(* Logix 5000 project; controller Modbus_TCP_Client_Example vendor 1 type 14 code 154 rev 32.15; software revision 32.05; part 2 of 10 *)

ADD_ON_INSTRUCTION AMP_Alarm_Reset_Servo   (* revision 1.0, vendor Applied Motion Products Inc. *)
// Applied Motion - Motor Alarm Reset - AOI
// Help:
// This AOI Reset Active Alarms(AX).
VAR_IN_OUT
   Input : DINT[20]; {required}   // Drive Input Assembly
   Output : DINT[11]; {required}   // Drive Output Assembly
        [10]   // Reserved
        [4]   // Target Velocity
        [0]   // Control Word
        [3]   // Target Pos
        [1]   // OpCode 1
        [2]   // OpCode 2
        [5]   // Porifle Acceleration
        [6]   // Profile Deceleration
        [7]   // Target Torque
        [8]   // OpCode 3
        [9]   // OpCode 4
END_VAR
VAR_INPUT
   Reset : BOOL; {required}   // Reset the Drive (on rising edge)
END_VAR
VAR_OUTPUT
   Sent : BOOL; {access Read Only, visible}   // Reset the Drive has been sent to drive
   In_Progress : BOOL; {access Read Only, visible}   // Reset in progress(not used)
   Done : BOOL; {access Read Only, visible}   // Reset completed without errors
   Error : BOOL; {access Read Only, visible}   // Reset failed
   State : DINT := 10; {access Read Only}   // Internal state of progress
END_VAR
VAR
   Loc_StatusCode : AMP_Status_Word_Servo; {access None}
   Loc_Reset_ONS : BOOL;
   Loc_Input_Assembly : AMP_Input_Assembly_Servo_v2; {access None}
   Loc_Command_Timeout : TIMER := (PRE := 2000); {access None}   // Timer to output fault if command is not Done
END_VAR

ROUTINE Logic   (* ladder *)
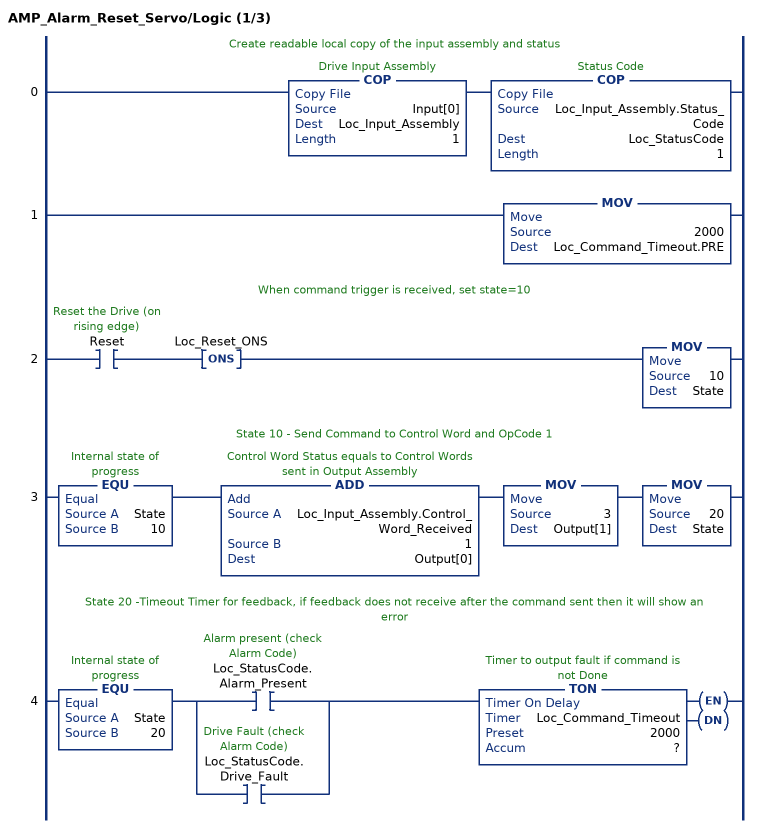
   // Create readable local copy of the input assembly and status
   0: COP(Input[0],Loc_Input_Assembly,1)COP(Loc_Input_Assembly.Status_Code,Loc_StatusCode,1);
   1: MOV(2000,Loc_Command_Timeout.PRE);
   // When command trigger is received, set state=10
   2: XIC(Reset)ONS(Loc_Reset_ONS)MOV(10,State);
   // State 10 - Send Command to Control Word and OpCode 1
   3: EQU(State,10)ADD(Loc_Input_Assembly.Control_Word_Received,1,Output[0])MOV(3,Output[1])MOV(20,State);
   // State 20 -Timeout Timer for feedback, if feedback does not receive after the command sent then it will show an error
   4: EQU(State,20)[XIC(Loc_StatusCode.Alarm_Present) ,XIC(Loc_StatusCode.Drive_Fault) ]TON(Loc_Command_Timeout,?,?);
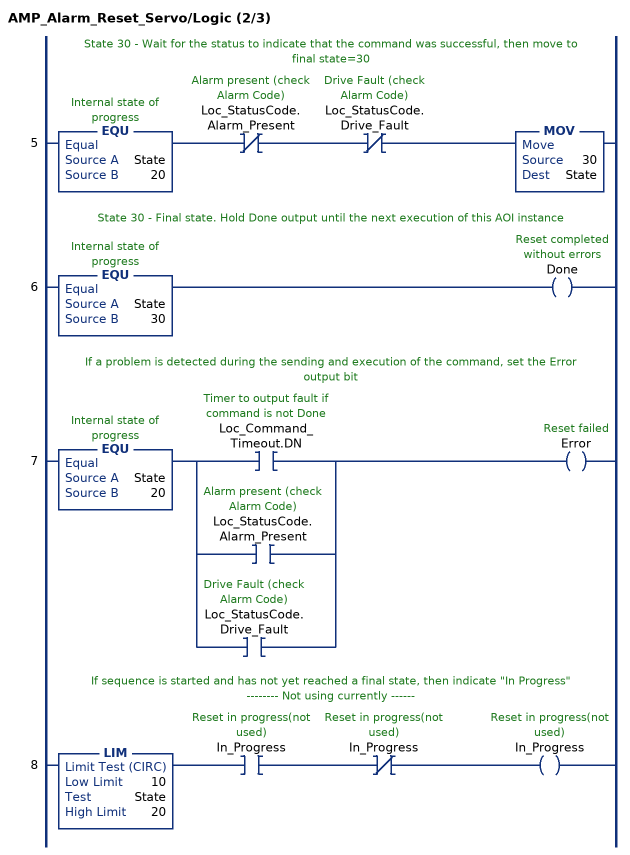
   // State 30 - Wait for the status to indicate that the command was successful, then move to final state=30
   5: EQU(State,20)XIO(Loc_StatusCode.Alarm_Present)XIO(Loc_StatusCode.Drive_Fault)MOV(30,State);
   // State 30 - Final state. Hold Done output until the next execution of this AOI instance
   6: EQU(State,30)OTE(Done);
   // If a problem is detected during the sending and execution of the command, set the Error output bit
   7: EQU(State,20)[XIC(Loc_Command_Timeout.DN) ,XIC(Loc_StatusCode.Alarm_Present) ,XIC(Loc_StatusCode.Drive_Fault) ]OTE(Error);
   // If sequence is started and has not yet reached a final state, then indicate "In Progress"
   // -------- Not using currently ------
   8: LIM(10,State,20)XIC(In_Progress)XIO(In_Progress)OTE(In_Progress);
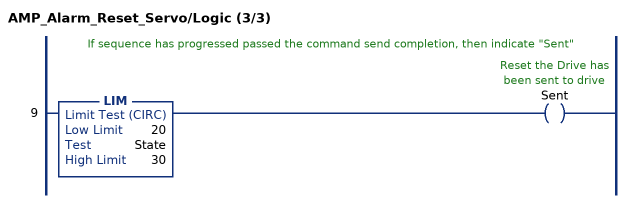
   // If sequence has progressed passed the command send completion, then indicate "Sent"
   9: LIM(20,State,30)OTE(Sent);
END_ROUTINE
END_ADD_ON_INSTRUCTION

ADD_ON_INSTRUCTION AMP_Crash_Stop_Servo   (* revision 1.0, vendor Applied Motion Products Inc. *)
// Applied Motion - Stop/Kill using Maximum Deceleration - AOI
// Help:
// This AOI immediately Stop the Motor Jogging/Moving(SK).
VAR_IN_OUT
   Input : DINT[20]; {required}   // Drive Input Assembly
        [4]   // Alarm_Code
        [16]   // Analog_Input1
        [0]   // Control_Word_Received
        [10]   // Position_Error
        [11]   // Actual_Velocity_RPS
        [12]   // Digital_Outputs
        [13]   // Digital_Inputs
        [14]   // Analog_Output1
        [15]   // Analog_Output2
        [17]   // Analog_Input2
        [18]   // Torque_Limit
        [19]   // Second_Encoder_Speed
        [1]   // OpCode1_Received
        [2]   // Control_Mode
        [3]   // Status_Code
        [5]   // Supply_Voltage
        [6]   // Applied_Torque
        [7]   // Drive_Temperature
        [8]   // Encoder_Position
        [9]   // Second_Encoder_Position
   Output : DINT[11]; {required}   // Drive Output Assembly
        [10]   // Reserved
        [4]   // Target Velocity
        [0]   // Control Word
        [3]   // Target Pos
        [1]   // OpCode 1
        [2]   // OpCode 2
        [5]   // Porifle Acceleration
        [6]   // Profile Deceleration
        [7]   // Target Torque
        [8]   // OpCode 3
        [9]   // OpCode 4
END_VAR
VAR_INPUT
   Stop : BOOL; {required}   // Crash Stop the drive axis (on rising edge)
END_VAR
VAR_OUTPUT
   Sent : BOOL; {access Read Only, visible}   // Stop has been sent to drive
   In_Progress : BOOL; {access Read Only, visible}   // Stop in progress
   Done : BOOL; {access Read Only, visible}   // Stop completed without errors - Servo is not moving
   Error : BOOL; {access Read Only, visible}   // Stop failed - drive not stopped or faulted
   State : DINT := 10; {access Read Only}   // Internal state of progress
END_VAR
VAR
   Loc_Stop_ONS : BOOL;
   Loc_StatusCode : AMP_Status_Word_Servo; {access None}
   Loc_Input_Assembly : AMP_Input_Assembly_Servo_v2; {access None}
END_VAR

ROUTINE Logic   (* ladder *)
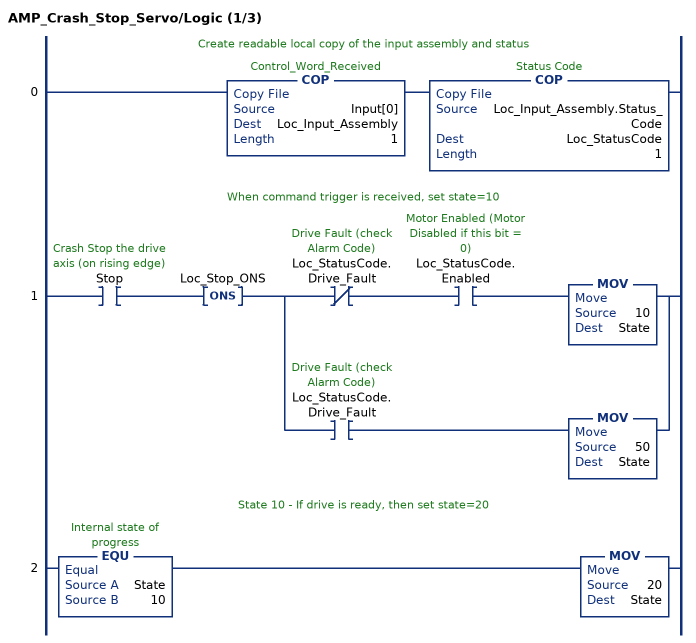
   // Create readable local copy of the input assembly and status
   0: COP(Input[0],Loc_Input_Assembly,1)COP(Loc_Input_Assembly.Status_Code,Loc_StatusCode,1);
   // When command trigger is received, set state=10
   1: XIC(Stop)ONS(Loc_Stop_ONS)[XIO(Loc_StatusCode.Drive_Fault) XIC(Loc_StatusCode.Enabled) MOV(10,State) ,XIC(Loc_StatusCode.Drive_Fault) MOV(50,State) ];
   // State 10 - If drive is ready, then set state=20
   2: EQU(State,10)MOV(20,State);
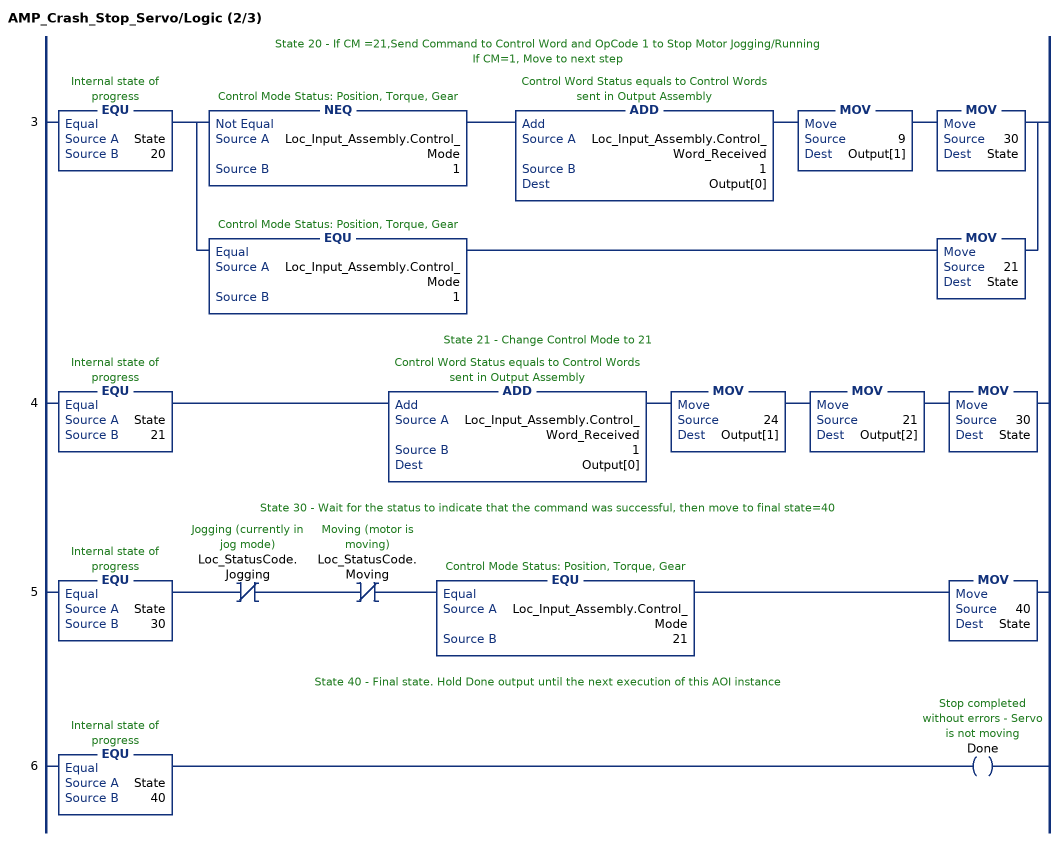
   // State 20 - If CM =21,Send Command to Control Word and OpCode 1 to Stop Motor Jogging/Running
   // If CM=1, Move to next step
   3: EQU(State,20)[NEQ(Loc_Input_Assembly.Control_Mode,1) ADD(Loc_Input_Assembly.Control_Word_Received,1,Output[0]) MOV(9,Output[1]) MOV(30,State) ,EQU(Loc_Input_Assembly.Control_Mode,1) MOV(21,State) ];
   // State 21 - Change Control Mode to 21
   4: EQU(State,21)ADD(Loc_Input_Assembly.Control_Word_Received,1,Output[0])MOV(24,Output[1])MOV(21,Output[2])MOV(30,State);
   // State 30 - Wait for the status to indicate that the command was successful, then move to final state=40
   5: EQU(State,30)XIO(Loc_StatusCode.Jogging)XIO(Loc_StatusCode.Moving)EQU(Loc_Input_Assembly.Control_Mode,21)MOV(40,State);
   // State 40 - Final state. Hold Done output until the next execution of this AOI instance
   6: EQU(State,40)OTE(Done);
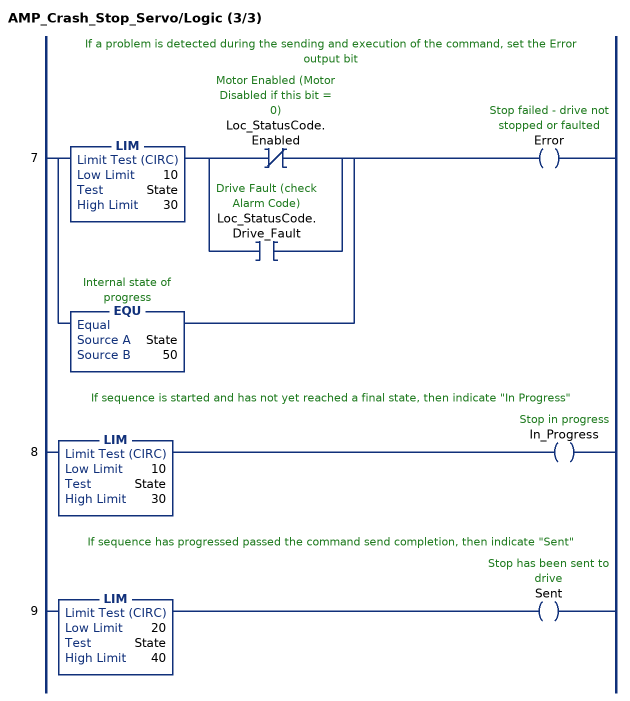
   // If a problem is detected during the sending and execution of the command, set the Error output bit
   7: [LIM(10,State,30) [XIO(Loc_StatusCode.Enabled) ,XIC(Loc_StatusCode.Drive_Fault) ] ,EQU(State,50) ]OTE(Error);
   // If sequence is started and has not yet reached a final state, then indicate "In Progress"
   8: LIM(10,State,30)OTE(In_Progress);
   // If sequence has progressed passed the command send completion, then indicate "Sent"
   9: LIM(20,State,40)OTE(Sent);
END_ROUTINE
END_ADD_ON_INSTRUCTION

ADD_ON_INSTRUCTION AMP_DI_Monitor_Servo   (* revision 1.0, vendor Applied Motion Products Inc. *)
// This AOI Monitor available Digital Input Status
// Help:
// Depending on which Drive/Motor Model you have, the number of IO Changes, Ignore extra IO monitoring
// 1 Represent Off/Open, 0 Represent On/Close
VAR_IN_OUT
   Input : DINT[20]; {required}   // Drive Input Assembly
END_VAR
VAR_OUTPUT
   DI_1 : BOOL; {visible}   // Digital Input 1, On = Input Opened, Off = Input Closed
   DI_2 : BOOL; {visible}   // Digital Input 2, On = Input Opened, Off = Input Closed
   DI_3 : BOOL; {visible}   // Digital Input 3, On = Input Opened, Off = Input Closed
   DI_4 : BOOL; {visible}   // Digital Input 4, On = Input Opened, Off = Input Closed
   DI_5 : BOOL; {visible}   // Digital Input 5, On = Input Opened, Off = Input Closed
   DI_6 : BOOL; {visible}   // Digital Input 6, On = Input Opened, Off = Input Closed
   DI_7 : BOOL; {visible}   // Digital Input 7, On = Input Opened, Off = Input Closed
   DI_8 : BOOL; {visible}   // Digital Input 8, On = Input Opened, Off = Input Closed
END_VAR
VAR
   Loc_StatusCode : AMP_Status_Word_Servo; {access None}
   Loc_Input_Assembly : AMP_Input_Assembly_Servo_v2; {access None}
   Inputs_DI : DINT; {access None}
END_VAR

ROUTINE Logic   (* ladder *)
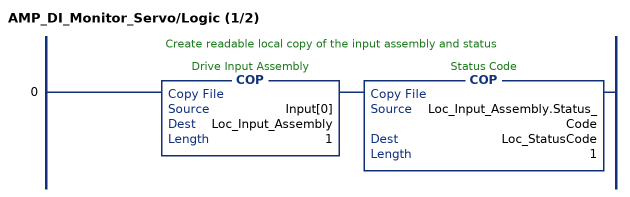
   // Create readable local copy of the input assembly and status
   0: COP(Input[0],Loc_Input_Assembly,1)COP(Loc_Input_Assembly.Status_Code,Loc_StatusCode,1);
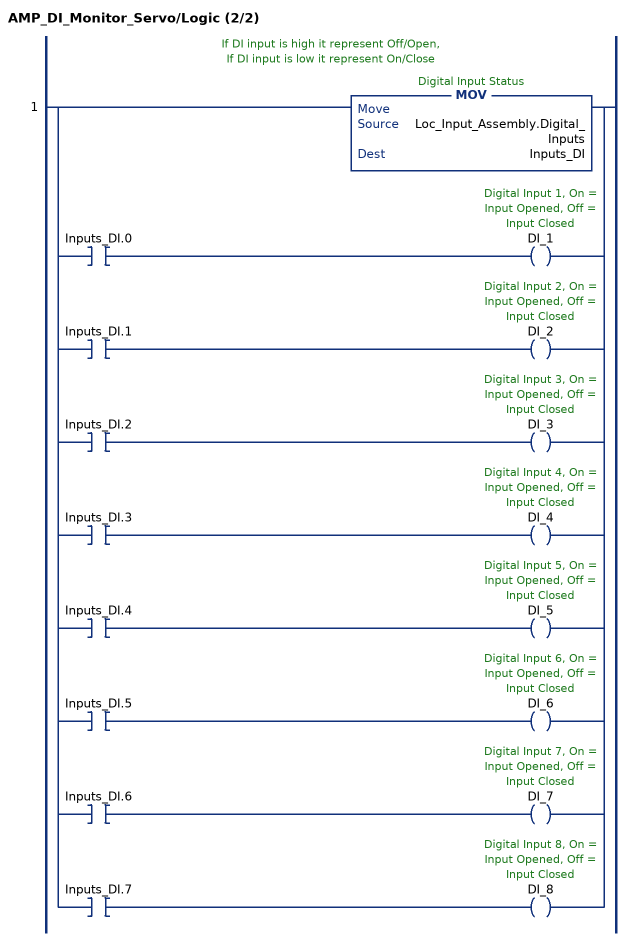
   // If DI input is high it represent Off/Open,
   // If DI input is low it represent On/Close
   1: [MOV(Loc_Input_Assembly.Digital_Inputs,Inputs_DI) ,XIC(Inputs_DI.0) OTE(DI_1) ,XIC(Inputs_DI.1) OTE(DI_2) ,XIC(Inputs_DI.2) OTE(DI_3) ,XIC(Inputs_DI.3) OTE(DI_4) ,XIC(Inputs_DI.4) OTE(DI_5) ,XIC(Inputs_DI.5) OTE(DI_6) ,XIC(Inputs_DI.6) OTE(DI_7) ,XIC(Inputs_DI.7) OTE(DI_8) ];
END_ROUTINE
END_ADD_ON_INSTRUCTION

ADD_ON_INSTRUCTION AMP_DO_Control_Servo   (* revision 1.0, vendor Applied Motion Products Inc. *)
// Applied Motion - General Purpose Digital Output Control - AOI
// Help:
// This AOI only Controls Output that are defined as General Purpose Output.
// Depending on which Drive/Motor Model you have, the number of Output Changes, Ignore extra Output.
// Define output number 1-6 and Condition L to Close the output, H to Open the Output.
// As an example, 2L will set output number 2 Close.
// This AOI can be used when Motor is Enable or Disable.
VAR_IN_OUT
   Input : DINT[20]; {required}   // Drive Input Assembly
        [16]   // Analog_Input1
        [4]   // Alarm_Code
        [0]   // Control_Word_Received
        [10]   // Position_Error
        [11]   // Actual_Velocity_RPS
        [12]   // Digital_Outputs
        [13]   // Digital_Inputs
        [14]   // Analog_Output1
        [15]   // Analog_Output2
        [17]   // Analog_Input2
        [18]   // Torque_Limit
        [19]   // Second_Encoder_Speed
        [1]   // OpCode1_Received
        [2]   // Control_Mode
        [3]   // Status_Code
        [5]   // Supply_Voltage
        [6]   // Applied_Torque
        [7]   // Drive_Temperature
        [8]   // Encoder_Position
        [9]   // Second_Encoder_Position
   Output : DINT[11]; {required}   // Drive Output Assembly
        [10]   // Reserved
        [4]   // Target Velocity
        [0]   // Control Word
        [3]   // Target Pos
        [1]   // OpCode 1
        [2]   // OpCode 2
        [5]   // Porifle Acceleration
        [6]   // Profile Deceleration
        [7]   // Target Torque
        [8]   // OpCode 3
        [9]   // OpCode 4
END_VAR
VAR_INPUT
   Execute : BOOL; {required}   // Execute the SCL command 'SO'
   Output_Number : INT; {required}   // Output Number, 1-6
   Condition : SINT; {required}   // Output Condition: H for Open and L for Close Output
END_VAR
VAR_OUTPUT
   DO_1 : BOOL; {visible}   // Digital Output 1, On = Output Closed, Off = Output Opened
   DO_2 : BOOL; {visible}   // Digital Output 2, On = Output Closed, Off = Output Opened
   DO_3 : BOOL; {visible}   // Digital Output 3, On = Output Closed, Off = Output Opened
   DO_4 : BOOL; {visible}   // Digital Output 4, On = Output Closed, Off = Output Opened
   DO_5 : BOOL; {visible}   // Digital Output 5, On = Output Closed, Off = Output Opened
   DO_6 : BOOL; {visible}   // Digital Output 6, On = Output Closed, Off = Output Opened
END_VAR
VAR
   Loc_StatusCode : AMP_Status_Word_Servo;
   Loc_Input_Assembly : AMP_Input_Assembly_Servo_v2;
   Loc_SCL_ONS : BOOL;
   Loc_Outputs_DO : INT; {access None}
   Loc_IO_Condition_Encoded : DINT; {access None}
   Loc_IO1_Number_Encoded : DINT; {access None}
   Loc_State : DINT := 10; {access Read Only}   // Internal state of progress
   Loc_Error : BOOL; {access Read Only}   // Command failed
   Loc_Done : BOOL; {access Read Only}   // Command completed without errors - Drive is Homed
   Loc_In_Progress : BOOL; {access Read Only}   // Command in progress
   Loc_Sent : BOOL; {access Read Only}   // Command has sent
END_VAR

ROUTINE Logic   (* ladder *)
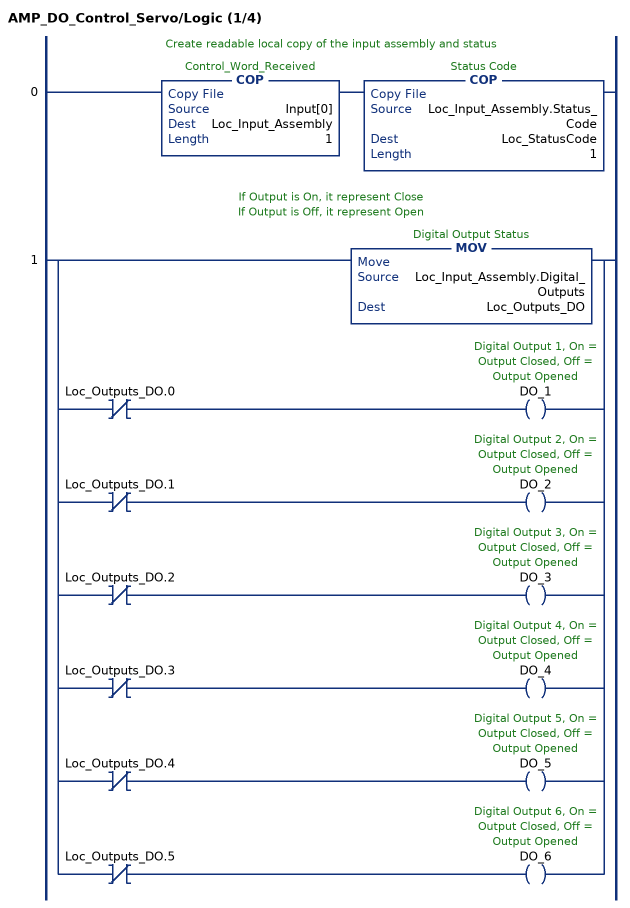
   // Create readable local copy of the input assembly and status
   0: COP(Input[0],Loc_Input_Assembly,1)COP(Loc_Input_Assembly.Status_Code,Loc_StatusCode,1);
   // If Output is On, it represent Close
   // If Output is Off, it represent Open
   1: [MOV(Loc_Input_Assembly.Digital_Outputs,Loc_Outputs_DO) ,XIO(Loc_Outputs_DO.0) OTE(DO_1) ,XIO(Loc_Outputs_DO.1) OTE(DO_2) ,XIO(Loc_Outputs_DO.2) OTE(DO_3) ,XIO(Loc_Outputs_DO.3) OTE(DO_4) ,XIO(Loc_Outputs_DO.4) OTE(DO_5) ,XIO(Loc_Outputs_DO.5) OTE(DO_6) ];
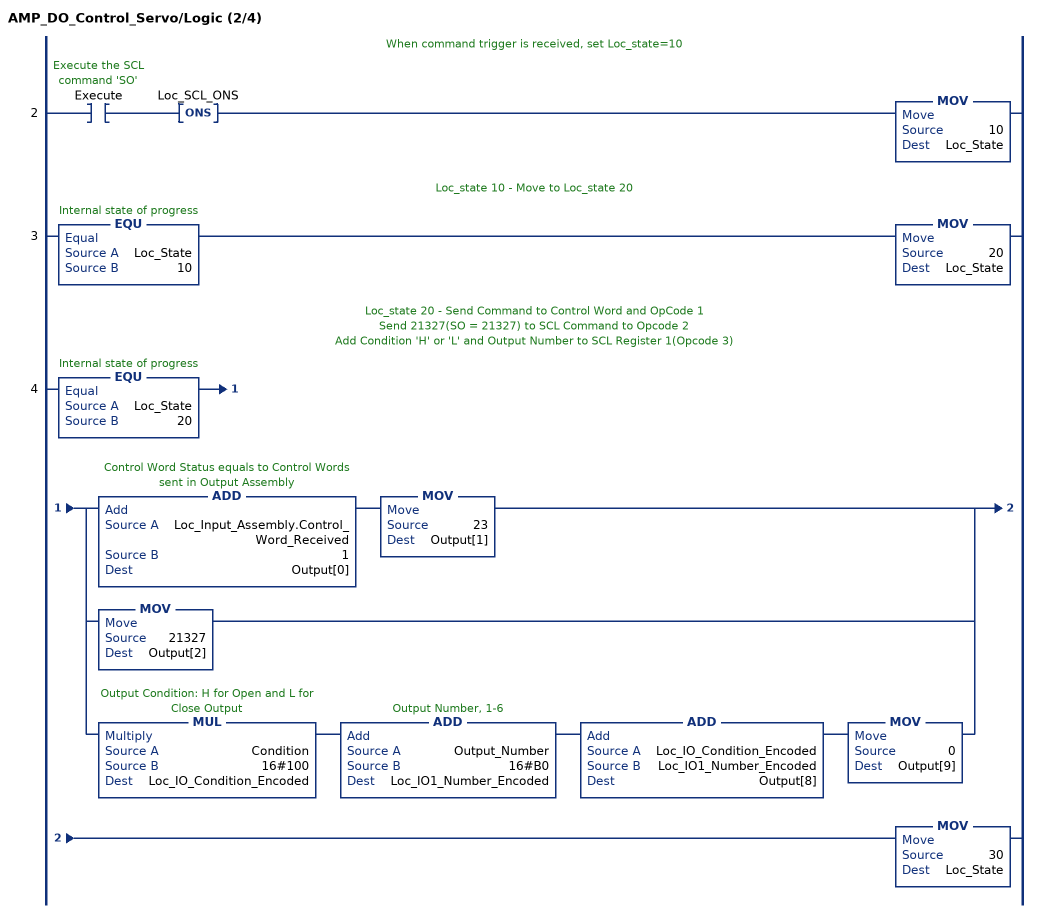
   // When command trigger is received, set Loc_state=10
   2: XIC(Execute)ONS(Loc_SCL_ONS)MOV(10,Loc_State);
   // Loc_state 10 - Move to Loc_state 20
   3: EQU(Loc_State,10)MOV(20,Loc_State);
   // Loc_state 20 - Send Command to Control Word and OpCode 1
   // Send 21327(SO = 21327) to SCL Command to Opcode 2
   // Add Condition 'H' or 'L' and Output Number to SCL Register 1(Opcode 3)
   4: EQU(Loc_State,20)[ADD(Loc_Input_Assembly.Control_Word_Received,1,Output[0]) MOV(23,Output[1]) ,MOV(21327,Output[2]) ,MUL(Condition,16#100,Loc_IO_Condition_Encoded) ADD(Output_Number,16#B0,Loc_IO1_Number_Encoded) ADD(Loc_IO_Condition_Encoded,Loc_IO1_Number_Encoded,Output[8]) MOV(0,Output[9]) ]MOV(30,Loc_State);
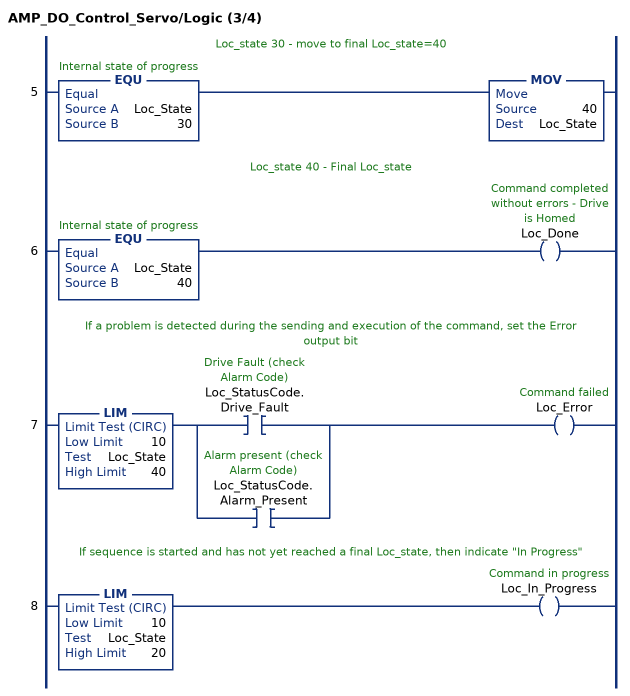
   // Loc_state 30 - move to final Loc_state=40
   5: EQU(Loc_State,30)MOV(40,Loc_State);
   // Loc_state 40 - Final Loc_state
   6: EQU(Loc_State,40)OTE(Loc_Done);
   // If a problem is detected during the sending and execution of the command, set the Error output bit
   7: LIM(10,Loc_State,40)[XIC(Loc_StatusCode.Drive_Fault) ,XIC(Loc_StatusCode.Alarm_Present) ]OTE(Loc_Error);
   // If sequence is started and has not yet reached a final Loc_state, then indicate "In Progress"
   8: LIM(10,Loc_State,20)OTE(Loc_In_Progress);
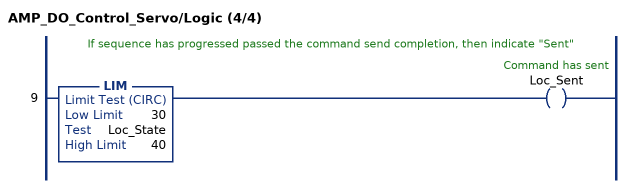
   // If sequence has progressed passed the command send completion, then indicate "Sent"
   9: LIM(30,Loc_State,40)OTE(Loc_Sent);
END_ROUTINE
END_ADD_ON_INSTRUCTION

ADD_ON_INSTRUCTION AMP_Hard_Stop_Homing   (* revision 1.0 *)
// Applied Motion - Hard Stop Homing AOI
// Help:
// The Hard Stop Homing AOI accepts all the required parameters for SCL commands HV1, HV2, HV3, HA1, HA2, HA3, HL1, HL2, HL3, HC, HD, HO and then sends the HS command to initiate the Hard Stop Homing move.
VAR_IN_OUT
   Input : DINT[14]; {required}   // Drive Input Assembly
   Output : DINT[16]; {required}   // Drive Output Assembly
        [0]   // Command Word
        [10]   // Data/Register 1
        [11]   // Data/Register 2
        [1]   // Jog Speed (0.25 rev/min)
        [2]   // Jog Acceleration (10 rev/s/s)
        [3]   // Jog Deceleration (10 rev/s/s)
        [4]   // Point-to-Point Velocity (0.25 rev/min)
        [5]   // Point-to-Point Acceleration (10 rev/s/s)
        [6]   // Point-to-Point Deceleration (10 rev/s/s)
        [7]   // Point-to-Point Distance (Motor steps)
        [9]   // (2x ASCII Letters in 16 lower word)
END_VAR
VAR_INPUT
   RPI : DINT := 100; {visible}   // Drive Connection Request Packet Interval (milliseconds)
   Start : BOOL; {required}   // Start the Homing
   HV1 : REAL; {required}   // Velocity used while seeking the hard stop (rev/s)
   HV2 : REAL; {required}   // Velocity when moving offset distance set by HO (rev/s)
   HV3 : REAL; {required}   // Velocity when searching for encoder index if desired (rev/s)
   HA1 : REAL; {required}   // Accel used while seeking the hard stop (rev/s/s)
   HA2 : REAL; {required}   // Accel when moving offset distance set by HO (rev/s/s)
   HA3 : REAL; {required}   // Accel when searching for encoder index if desired (rev/s/s)
   HL1 : REAL; {required}   // Decel used while seeking the hard stop (rev/s/s)
   HL2 : REAL; {required}   // Decel when moving offset distance set by HO (rev/s/s)
   HL3 : REAL; {required}   // Decel when searching for encoder index if desired (rev/s/s)
   HC : REAL; {required}   // Hard Stop Current (Amps)
   HD : DINT; {required}   // Hard Stop Fault Delay (ms)
   HO : DINT; {required}   // Home Offset (steps, negative = CCW, positive = CW)
   HS : DINT; {required}   // Hard Stop method (0 = without index, 1 = with index)
END_VAR
VAR_OUTPUT
   Sent : BOOL; {access Read Only, visible}   // All parameter setting and homing commands have been sent to drive
   In_Progress : BOOL; {access Read Only, visible}   // The setting of parameters and/or homing are in progress
   Done : BOOL; {access Read Only, visible}   // Homing Move completed without errors - desired position reached
   Error : BOOL; {access Read Only, visible}   // Homing failed to complete - drive not ready or faulted
   State : DINT := 34; {access Read Only}   // Internal state of progress
END_VAR
VAR
   Loc_StatusCode : AMP_Status_Word;
   Loc_CommandOff_Timer : TIMER;   // Timer to make sure command value was 0 before sending a new command
   Loc_CommandOn_Timer : TIMER;   // Timer to make sure command value is set long enough to be sent to drive
   Loc_Input_Assembly : AMP_Input_Assembly_v2; {access None}
   Loc_Start_ONS : BOOL; {access None}
END_VAR

ROUTINE Logic   (* ladder *)
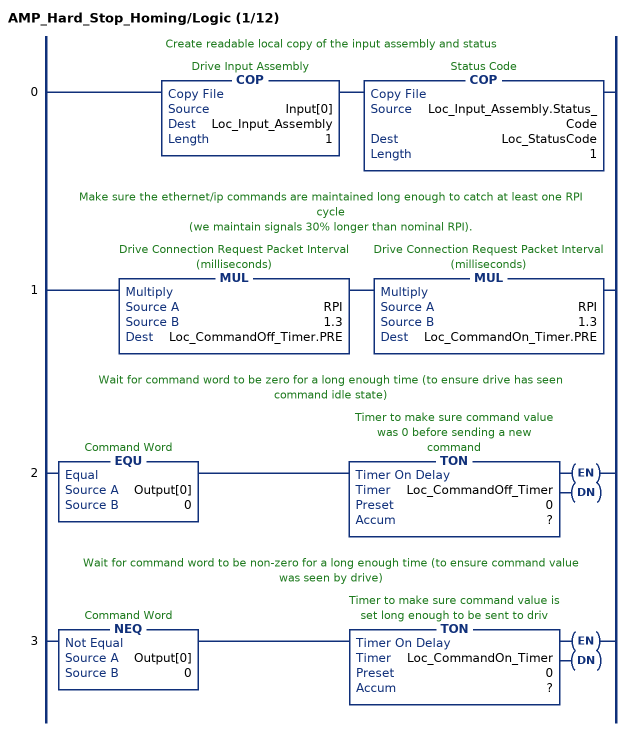
   // Create readable local copy of the input assembly and status
   0: COP(Input[0],Loc_Input_Assembly,1)COP(Loc_Input_Assembly.Status_Code,Loc_StatusCode,1);
   // Make sure the ethernet/ip commands are maintained long enough to catch at least one RPI cycle
   // (we maintain signals 30% longer than nominal RPI).
   1: MUL(RPI,1.3,Loc_CommandOff_Timer.PRE)MUL(RPI,1.3,Loc_CommandOn_Timer.PRE);
   // Wait for command word to be zero for a long enough time (to ensure drive has seen command idle state)
   2: EQU(Output[0],0)TON(Loc_CommandOff_Timer,?,?);
   // Wait for command word to be non-zero for a long enough time (to ensure command value was seen by drive)
   3: NEQ(Output[0],0)TON(Loc_CommandOn_Timer,?,?);
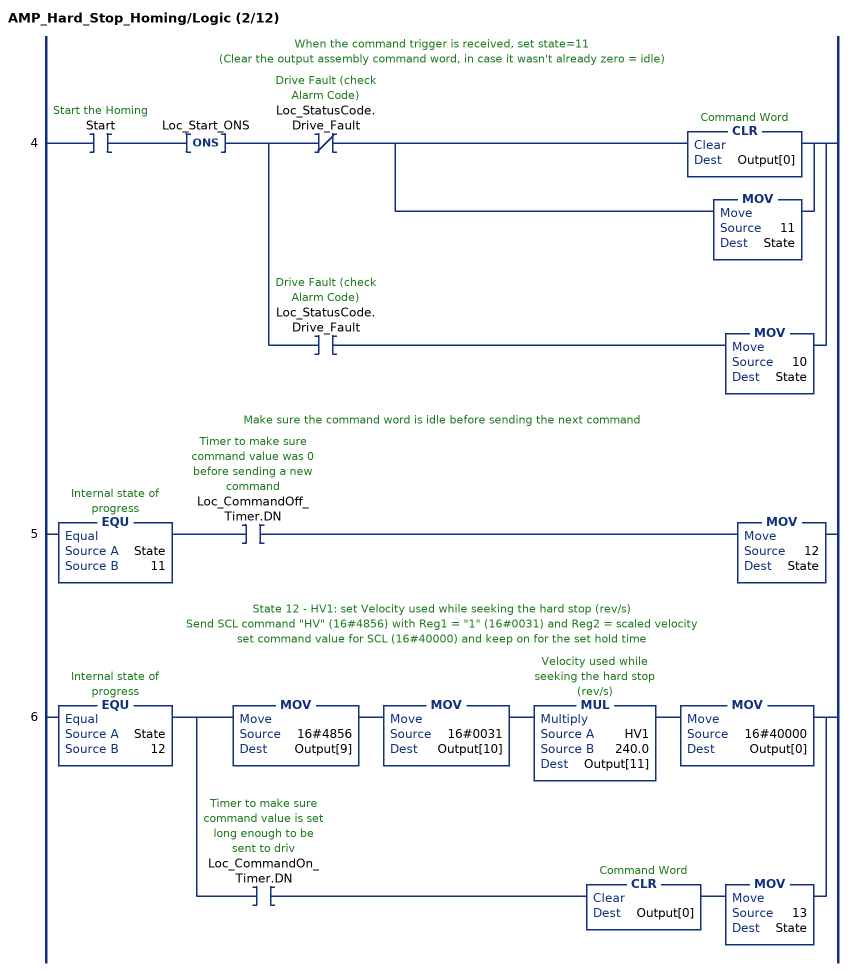
   // When the command trigger is received, set state=11
   // (Clear the output assembly command word, in case it wasn't already zero = idle)
   4: XIC(Start)ONS(Loc_Start_ONS)[XIO(Loc_StatusCode.Drive_Fault) [CLR(Output[0]) ,MOV(11,State) ] ,XIC(Loc_StatusCode.Drive_Fault) MOV(10,State) ];
   // Make sure the command word is idle before sending the next command
   5: EQU(State,11)XIC(Loc_CommandOff_Timer.DN)MOV(12,State);
   // State 12 - HV1: set Velocity used while seeking the hard stop (rev/s)
   // Send SCL command "HV" (16#4856) with Reg1 = "1" (16#0031) and Reg2 = scaled velocity
   // set command value for SCL (16#40000) and keep on for the set hold time
   6: EQU(State,12)[MOV(16#4856,Output[9]) MOV(16#0031,Output[10]) MUL(HV1,240.0,Output[11]) MOV(16#40000,Output[0]) ,XIC(Loc_CommandOn_Timer.DN) CLR(Output[0]) MOV(13,State) ];
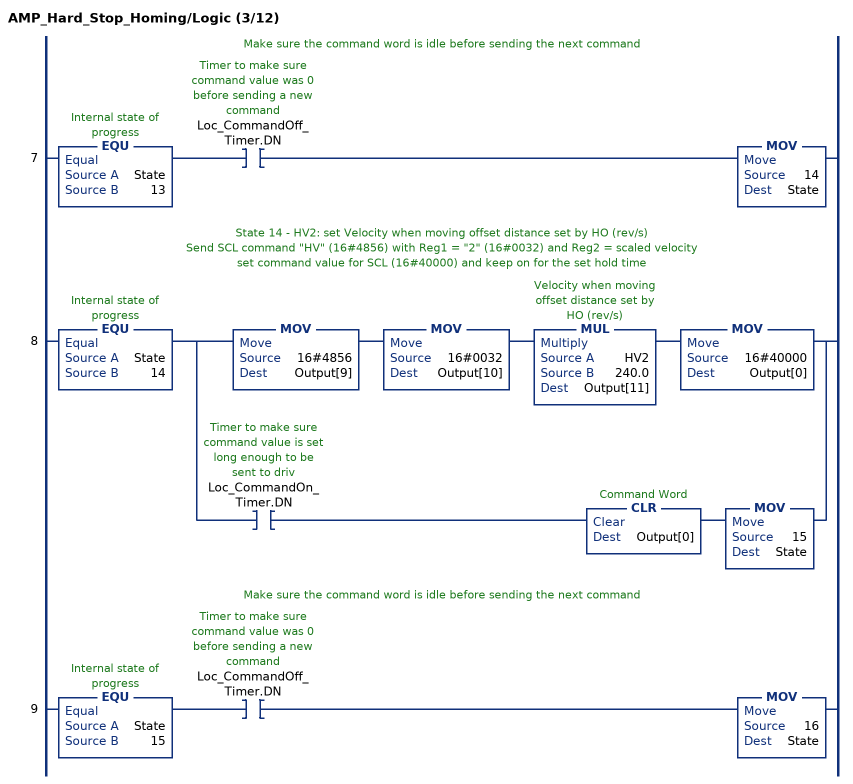
   // Make sure the command word is idle before sending the next command
   7: EQU(State,13)XIC(Loc_CommandOff_Timer.DN)MOV(14,State);
   // State 14 - HV2: set Velocity when moving offset distance set by HO (rev/s)
   // Send SCL command "HV" (16#4856) with Reg1 = "2" (16#0032) and Reg2 = scaled velocity
   // set command value for SCL (16#40000) and keep on for the set hold time
   8: EQU(State,14)[MOV(16#4856,Output[9]) MOV(16#0032,Output[10]) MUL(HV2,240.0,Output[11]) MOV(16#40000,Output[0]) ,XIC(Loc_CommandOn_Timer.DN) CLR(Output[0]) MOV(15,State) ];
   // Make sure the command word is idle before sending the next command
   9: EQU(State,15)XIC(Loc_CommandOff_Timer.DN)MOV(16,State);
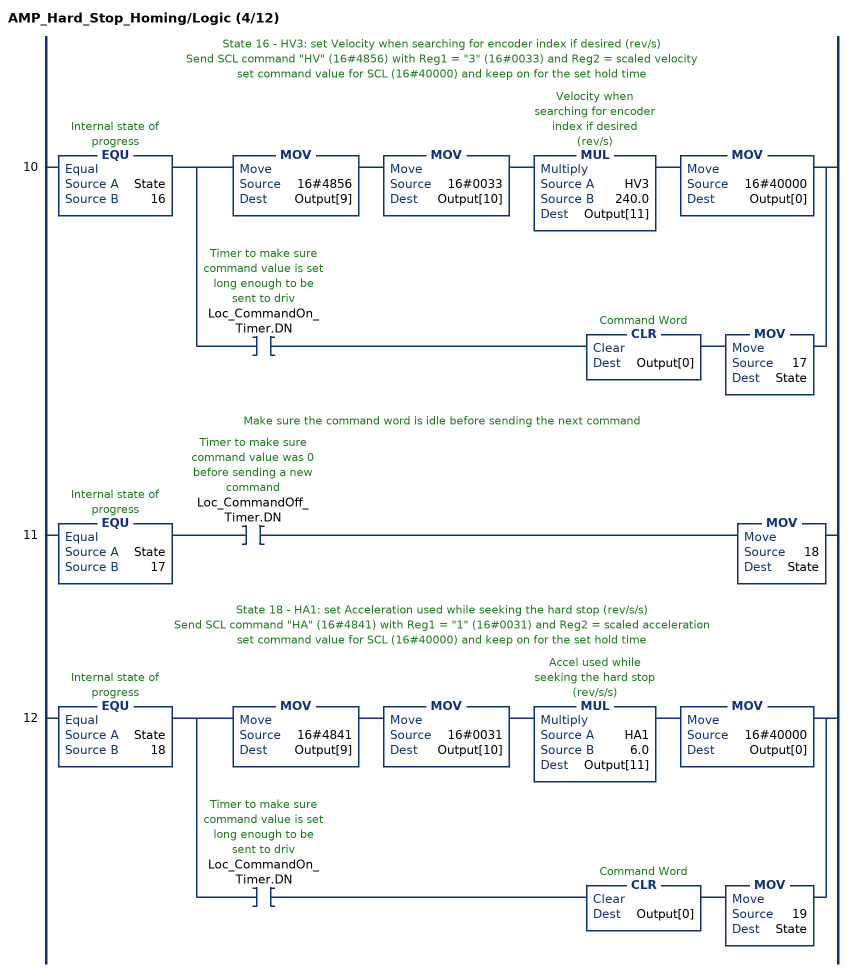
   // State 16 - HV3: set Velocity when searching for encoder index if desired (rev/s)
   // Send SCL command "HV" (16#4856) with Reg1 = "3" (16#0033) and Reg2 = scaled velocity
   // set command value for SCL (16#40000) and keep on for the set hold time
   10: EQU(State,16)[MOV(16#4856,Output[9]) MOV(16#0033,Output[10]) MUL(HV3,240.0,Output[11]) MOV(16#40000,Output[0]) ,XIC(Loc_CommandOn_Timer.DN) CLR(Output[0]) MOV(17,State) ];
   // Make sure the command word is idle before sending the next command
   11: EQU(State,17)XIC(Loc_CommandOff_Timer.DN)MOV(18,State);
   // State 18 - HA1: set Acceleration used while seeking the hard stop (rev/s/s)
   // Send SCL command "HA" (16#4841) with Reg1 = "1" (16#0031) and Reg2 = scaled acceleration
   // set command value for SCL (16#40000) and keep on for the set hold time
   12: EQU(State,18)[MOV(16#4841,Output[9]) MOV(16#0031,Output[10]) MUL(HA1,6.0,Output[11]) MOV(16#40000,Output[0]) ,XIC(Loc_CommandOn_Timer.DN) CLR(Output[0]) MOV(19,State) ];
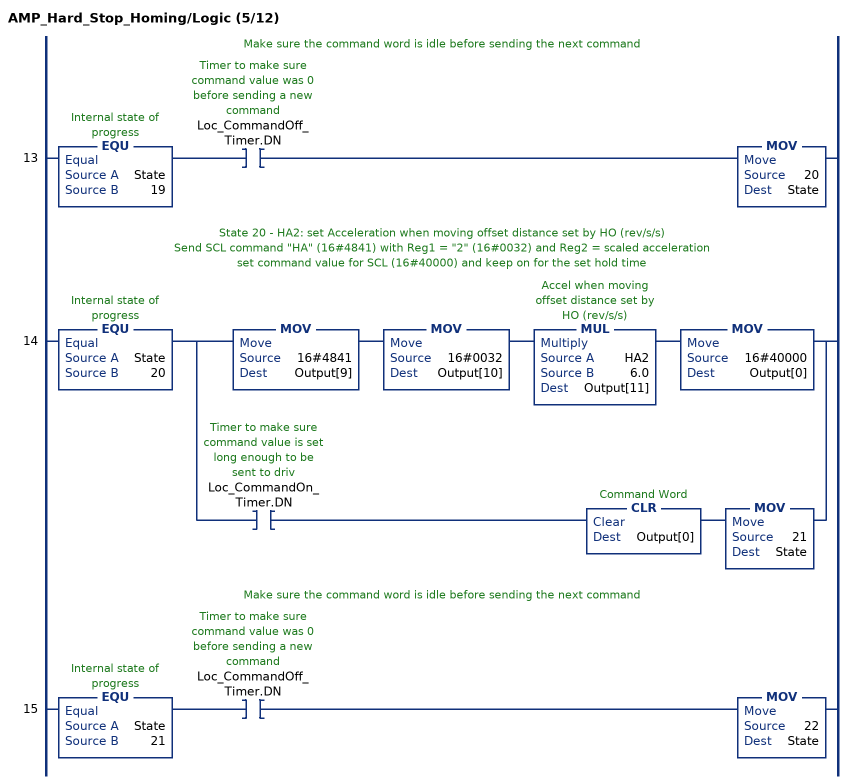
   // Make sure the command word is idle before sending the next command
   13: EQU(State,19)XIC(Loc_CommandOff_Timer.DN)MOV(20,State);
   // State 20 - HA2: set Acceleration when moving offset distance set by HO (rev/s/s)
   // Send SCL command "HA" (16#4841) with Reg1 = "2" (16#0032) and Reg2 = scaled acceleration
   // set command value for SCL (16#40000) and keep on for the set hold time
   14: EQU(State,20)[MOV(16#4841,Output[9]) MOV(16#0032,Output[10]) MUL(HA2,6.0,Output[11]) MOV(16#40000,Output[0]) ,XIC(Loc_CommandOn_Timer.DN) CLR(Output[0]) MOV(21,State) ];
   // Make sure the command word is idle before sending the next command
   15: EQU(State,21)XIC(Loc_CommandOff_Timer.DN)MOV(22,State);
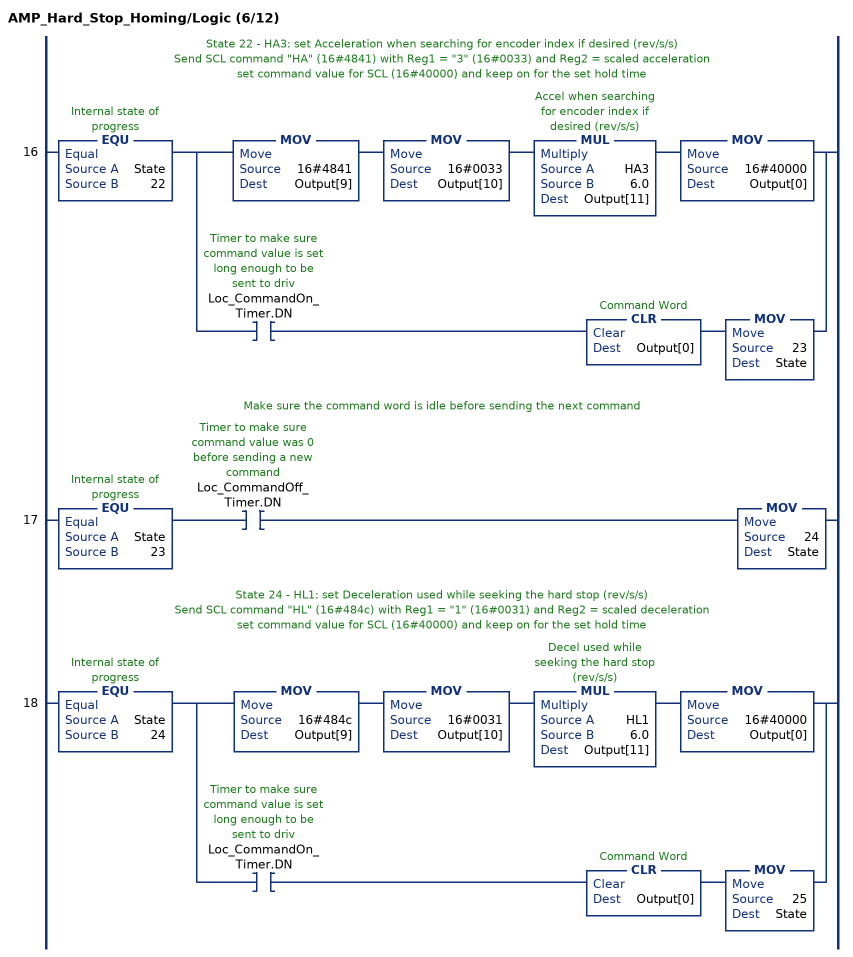
   // State 22 - HA3: set Acceleration when searching for encoder index if desired (rev/s/s)
   // Send SCL command "HA" (16#4841) with Reg1 = "3" (16#0033) and Reg2 = scaled acceleration
   // set command value for SCL (16#40000) and keep on for the set hold time
   16: EQU(State,22)[MOV(16#4841,Output[9]) MOV(16#0033,Output[10]) MUL(HA3,6.0,Output[11]) MOV(16#40000,Output[0]) ,XIC(Loc_CommandOn_Timer.DN) CLR(Output[0]) MOV(23,State) ];
   // Make sure the command word is idle before sending the next command
   17: EQU(State,23)XIC(Loc_CommandOff_Timer.DN)MOV(24,State);
   // State 24 - HL1: set Deceleration used while seeking the hard stop (rev/s/s)
   // Send SCL command "HL" (16#484c) with Reg1 = "1" (16#0031) and Reg2 = scaled deceleration
   // set command value for SCL (16#40000) and keep on for the set hold time
   18: EQU(State,24)[MOV(16#484c,Output[9]) MOV(16#0031,Output[10]) MUL(HL1,6.0,Output[11]) MOV(16#40000,Output[0]) ,XIC(Loc_CommandOn_Timer.DN) CLR(Output[0]) MOV(25,State) ];
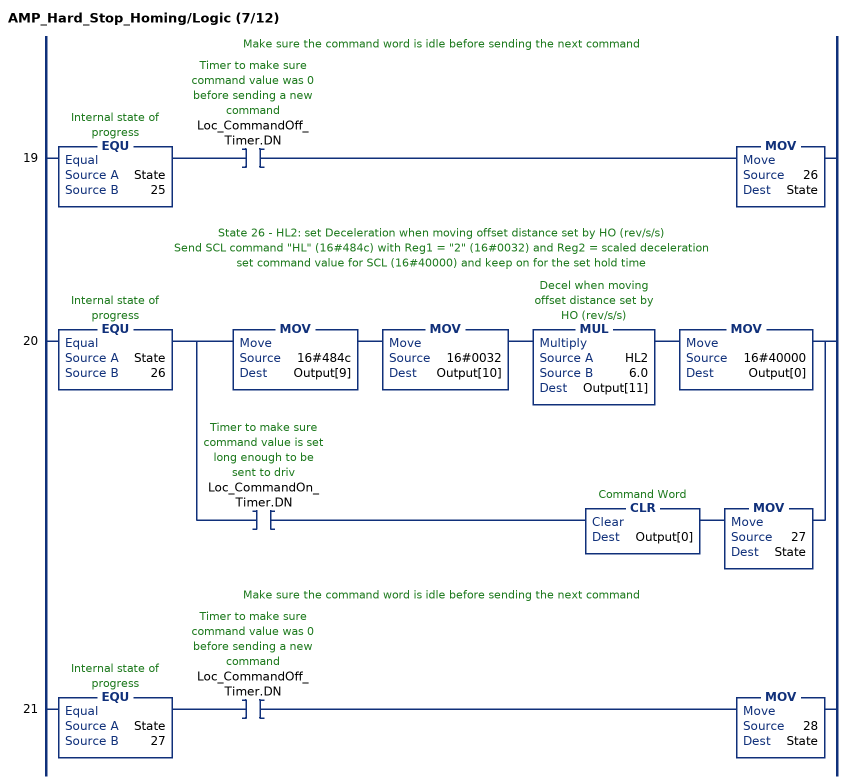
   // Make sure the command word is idle before sending the next command
   19: EQU(State,25)XIC(Loc_CommandOff_Timer.DN)MOV(26,State);
   // State 26 - HL2: set Deceleration when moving offset distance set by HO (rev/s/s)
   // Send SCL command "HL" (16#484c) with Reg1 = "2" (16#0032) and Reg2 = scaled deceleration
   // set command value for SCL (16#40000) and keep on for the set hold time
   20: EQU(State,26)[MOV(16#484c,Output[9]) MOV(16#0032,Output[10]) MUL(HL2,6.0,Output[11]) MOV(16#40000,Output[0]) ,XIC(Loc_CommandOn_Timer.DN) CLR(Output[0]) MOV(27,State) ];
   // Make sure the command word is idle before sending the next command
   21: EQU(State,27)XIC(Loc_CommandOff_Timer.DN)MOV(28,State);
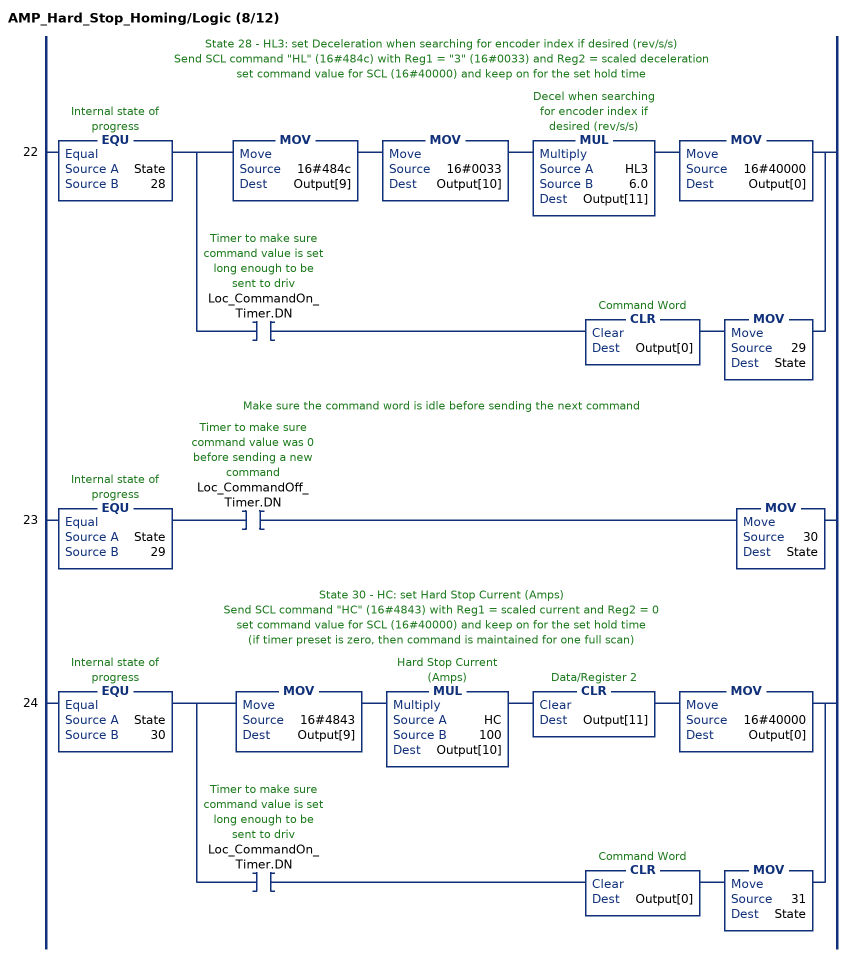
   // State 28 - HL3: set Deceleration when searching for encoder index if desired (rev/s/s)
   // Send SCL command "HL" (16#484c) with Reg1 = "3" (16#0033) and Reg2 = scaled deceleration
   // set command value for SCL (16#40000) and keep on for the set hold time
   22: EQU(State,28)[MOV(16#484c,Output[9]) MOV(16#0033,Output[10]) MUL(HL3,6.0,Output[11]) MOV(16#40000,Output[0]) ,XIC(Loc_CommandOn_Timer.DN) CLR(Output[0]) MOV(29,State) ];
   // Make sure the command word is idle before sending the next command
   23: EQU(State,29)XIC(Loc_CommandOff_Timer.DN)MOV(30,State);
   // State 30 - HC: set Hard Stop Current (Amps)
   // Send SCL command "HC" (16#4843) with Reg1 = scaled current and Reg2 = 0
   // set command value for SCL (16#40000) and keep on for the set hold time
   // (if timer preset is zero, then command is maintained for one full scan)
   24: EQU(State,30)[MOV(16#4843,Output[9]) MUL(HC,100,Output[10]) CLR(Output[11]) MOV(16#40000,Output[0]) ,XIC(Loc_CommandOn_Timer.DN) CLR(Output[0]) MOV(31,State) ];
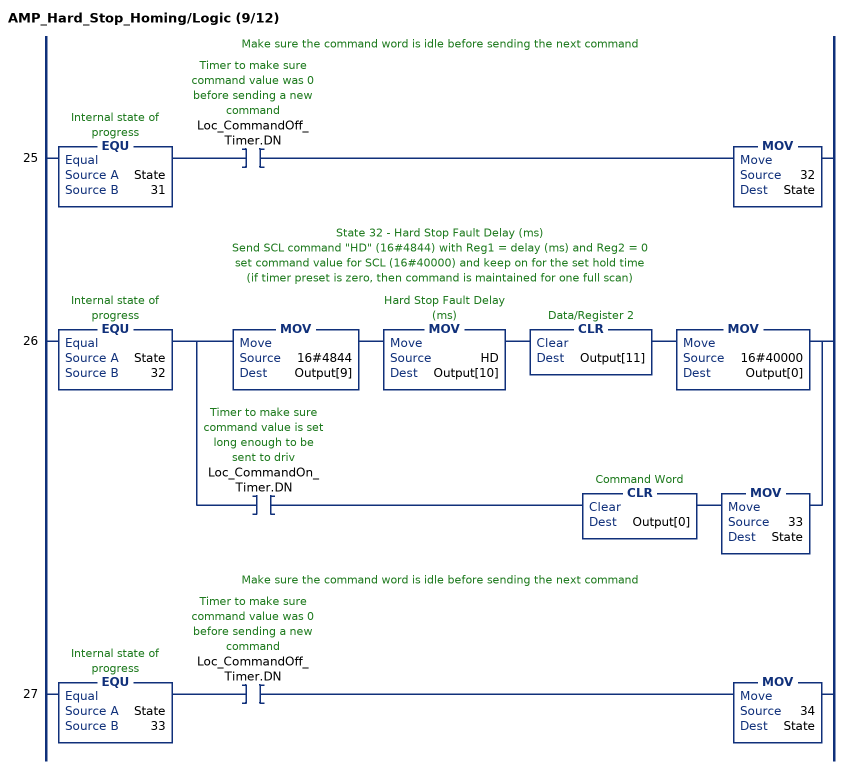
   // Make sure the command word is idle before sending the next command
   25: EQU(State,31)XIC(Loc_CommandOff_Timer.DN)MOV(32,State);
   // State 32 - Hard Stop Fault Delay (ms)
   // Send SCL command "HD" (16#4844) with Reg1 = delay (ms) and Reg2 = 0
   // set command value for SCL (16#40000) and keep on for the set hold time
   // (if timer preset is zero, then command is maintained for one full scan)
   26: EQU(State,32)[MOV(16#4844,Output[9]) MOV(HD,Output[10]) CLR(Output[11]) MOV(16#40000,Output[0]) ,XIC(Loc_CommandOn_Timer.DN) CLR(Output[0]) MOV(33,State) ];
   // Make sure the command word is idle before sending the next command
   27: EQU(State,33)XIC(Loc_CommandOff_Timer.DN)MOV(34,State);
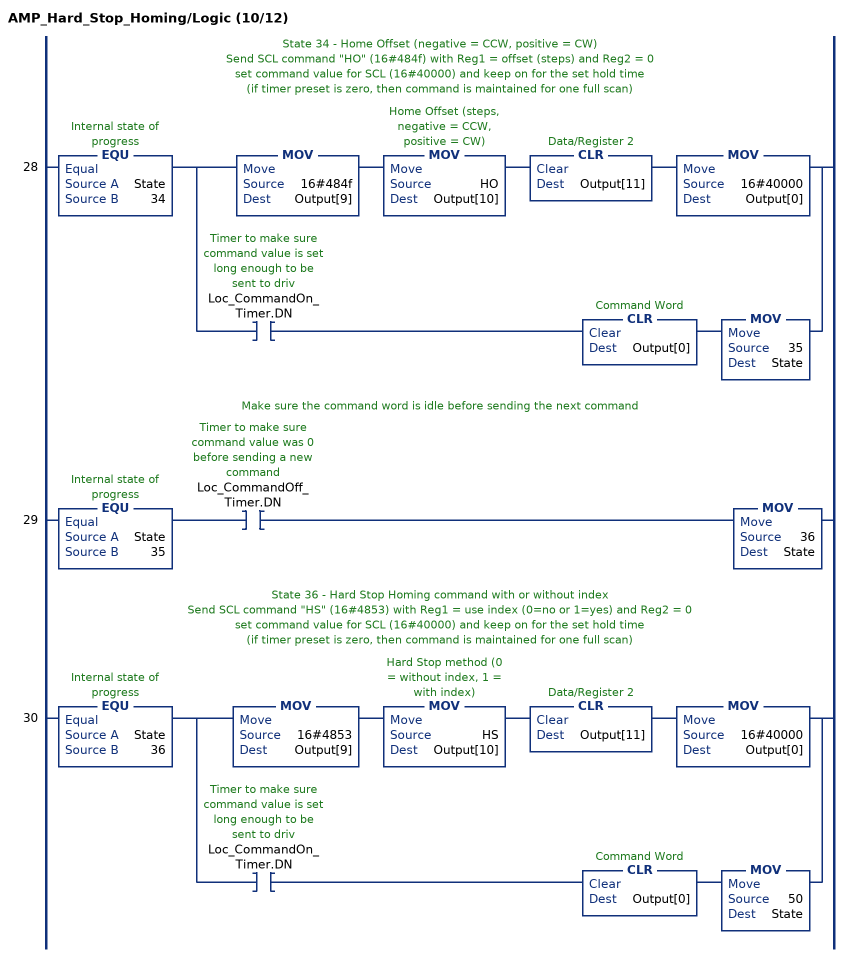
   // State 34 - Home Offset (negative = CCW, positive = CW)
   // Send SCL command "HO" (16#484f) with Reg1 = offset (steps) and Reg2 = 0
   // set command value for SCL (16#40000) and keep on for the set hold time
   // (if timer preset is zero, then command is maintained for one full scan)
   28: EQU(State,34)[MOV(16#484f,Output[9]) MOV(HO,Output[10]) CLR(Output[11]) MOV(16#40000,Output[0]) ,XIC(Loc_CommandOn_Timer.DN) CLR(Output[0]) MOV(35,State) ];
   // Make sure the command word is idle before sending the next command
   29: EQU(State,35)XIC(Loc_CommandOff_Timer.DN)MOV(36,State);
   // State 36 - Hard Stop Homing command with or without index
   // Send SCL command "HS" (16#4853) with Reg1 = use index (0=no or 1=yes) and Reg2 = 0
   // set command value for SCL (16#40000) and keep on for the set hold time
   // (if timer preset is zero, then command is maintained for one full scan)
   30: EQU(State,36)[MOV(16#4853,Output[9]) MOV(HS,Output[10]) CLR(Output[11]) MOV(16#40000,Output[0]) ,XIC(Loc_CommandOn_Timer.DN) CLR(Output[0]) MOV(50,State) ];
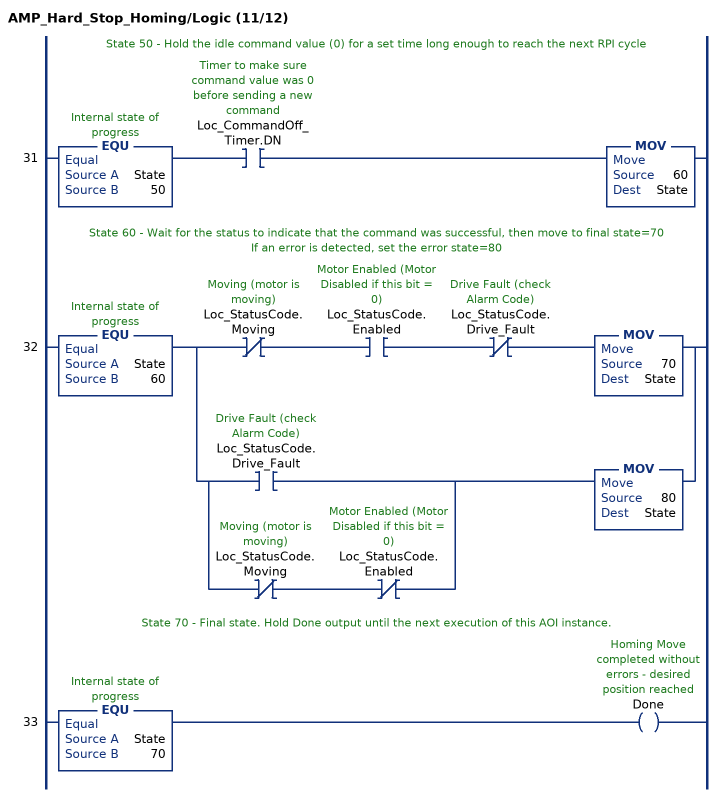
   // State 50 - Hold the idle command value (0) for a set time long enough to reach the next RPI cycle
   31: EQU(State,50)XIC(Loc_CommandOff_Timer.DN)MOV(60,State);
   // State 60 - Wait for the status to indicate that the command was successful, then move to final state=70
   // If an error is detected, set the error state=80
   32: EQU(State,60)[XIO(Loc_StatusCode.Moving) XIC(Loc_StatusCode.Enabled) XIO(Loc_StatusCode.Drive_Fault) MOV(70,State) ,[XIC(Loc_StatusCode.Drive_Fault) ,XIO(Loc_StatusCode.Moving) XIO(Loc_StatusCode.Enabled) ] MOV(80,State) ];
   // State 70 - Final state. Hold Done output until the next execution of this AOI instance.
   33: EQU(State,70)OTE(Done);
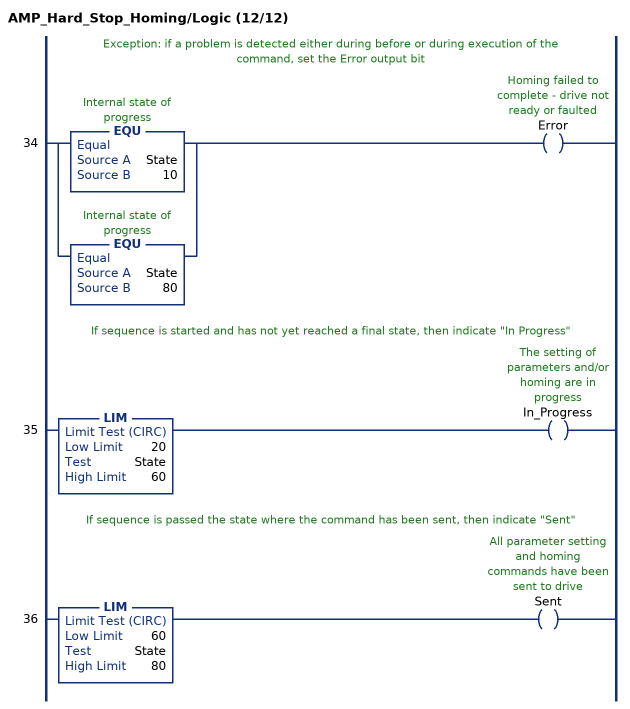
   // Exception: if a problem is detected either during before or during execution of the command, set the Error output bit
   34: [EQU(State,10) ,EQU(State,80) ]OTE(Error);
   // If sequence is started and has not yet reached a final state, then indicate "In Progress"
   35: LIM(20,State,60)OTE(In_Progress);
   // If sequence is passed the state where the command has been sent, then indicate "Sent"
   36: LIM(60,State,80)OTE(Sent);
END_ROUTINE
END_ADD_ON_INSTRUCTION
